(* PLC project Generated.project, CODESYS CODESYS V3.5 SP19 Patch 1 *)
(* stored: creationDateTime 2026-09-06T13:00:42.373519, modificationDateTime 2026-09-06T13:00:42.373519 *)

(* values of E_Diag_State: DISABLED: Désactivé (surveillance non active); READY: Opérationnel réel, pas de défaut; INIT: Initialisation / Recherche de réseau; MONITORING: Surveillance active (états transitoires); ERROR: Anomalie de communication; SIMULATED: Bypass simulation ou bypass réseau IHM — pas le bus réel *)

{attribute 'qualified_only'}
{attribute 'strict'}
TYPE E_Diag_State : (DISABLED := 0, READY := 1, INIT := 2, MONITORING := 3, ERROR := 4, SIMULATED := 5);
END_TYPE
